# EPICS autosave request: xxxApp/Db/Security_Control_settings.req
$(P)AS_OnOff
$(P)LocalAccess
$(P)RemoteAccess
